// TIA Portal V16 export
// export: Created 2024-12-03T15:41:40.0922187Z, ExportSetting WithDefaults, DisplayName Totally Integrated Automation Portal, DisplayVersion V16 Update 6, DisplayName TIA Portal Version Control Interface, DisplayVersion V16 Update 2, DisplayName TIA Portal Openness, DisplayVersion V16 Update 6, DisplayName TIA Portal Teamcenter Gateway, DisplayVersion V16, DisplayName SINAMICS Startdrive Advanced, DisplayVersion V16 Update 5, DisplayName SINAMICS Startdrive G130, G150, S120, S150, SINAMICS MV, S210, DisplayVersion V16 Update 5, DisplayName SINAMICS Startdrive G110M, G120, G120C, G120D, G120P, G115D, DisplayVersion V16 Update 5, DisplayName STEP 7 Professional, DisplayVersion V16 Update 6, DisplayName STEP 7 Safety, DisplayVersion V16, DisplayName WinCC Advanced / Unified PC, DisplayVersion V16 Update 6
FUNCTION_BLOCK "Settings_Conveyor_zone_Index_FB"   // FB77, SCL
{ S7_Optimized_Access := 'TRUE' }
VERSION : 0.1
// stored: AutoNumber true, IsIECCheckEnabled false, IsRetainMemResEnabled false, MemoryReserve 100, SetENOAutomatically false, UDAEnableTagReadback false
   VAR
      settingsSaved : Bool;
   END_VAR
BEGIN
   IF NOT #settingsSaved OR "HMI_DB".ReloadSettings.signal THEN
       #settingsSaved := true;

       REGION ZONE CONVEYORS

           "CONV_DB".CONV_101.Zone := 1;
           "CONV_DB".CONV_102L.Zone := 1;
           "CONV_DB".CONV_102R.Zone := 1;
           "CONV_DB".CONV_103L.Zone := 1;
           "CONV_DB".CONV_103R.Zone := 1;
           "CONV_DB".CONV_104L.Zone := 1;
           "CONV_DB".CONV_104R.Zone := 1;
           "CONV_DB".CONV_105L.Zone := 1;
           "CONV_DB".CONV_105R.Zone := 1;
           "CONV_DB".CONV_106R.Zone := 1;
           "CONV_DB".CONV_107R.Zone := 1;
           "CONV_DB".CONV_108L.Zone := 1;
           "CONV_DB".CONV_108R.Zone := 1;
           "CONV_DB".CONV_109L.Zone := 1;
           "CONV_DB".CONV_109R.Zone := 1;
           "CONV_DB".CONV_110L.Zone := 1;
           "CONV_DB".CONV_110R.Zone := 1;
           "CONV_DB".CONV_111L.Zone := 1;
           "CONV_DB".CONV_111R.Zone := 1;
           "CONV_DB".CONV_112R.Zone := 1;
           "CONV_DB".CONV_113L.Zone := 1;
           "CONV_DB".CONV_113R.Zone := 1;
           "CONV_DB".CONV_114L.Zone := 1;
           "CONV_DB".CONV_114R.Zone := 1;
           "CONV_DB".CONV_115L.Zone := 1;
           "CONV_DB".CONV_115R.Zone := 1;
           "CONV_DB".CONV_201R_BELTS.Zone := 1;
           "CONV_DB".CONV_203R_BELTS.Zone := 1;
           "CONV_DB".CONV_301R.Zone := 1;
           "CONV_DB".CONV_302L.Zone := 1;
           "CONV_DB".CONV_302R.Zone := 1;
           "CONV_DB".CONV_303L.Zone := 1;
           "CONV_DB".CONV_303R.Zone := 1;
           "CONV_DB".CONV_304L.Zone := 1;
           "CONV_DB".CONV_304R.Zone := 1;
           "CONV_DB".CONV_305R.Zone := 1;

           "Scanners_DB".SCAN_100.Zone := 1;

       END_REGION



   END_IF;
END_FUNCTION_BLOCK
